(* CODESYS project BallSorting_student1.project

Project tree, tasks and I/O mapping:
  Device : CODESYS Control Win V3, 3S - Smart Software Solutions GmbH, version 3.5.17.10
    application Application
      libraries: Standard, * (System); Util, * (System); VisuDialogs, * (System)
      task MainTask (cyclic, interval t#20ms, priority 1) calls Model, PLC_PRG
      program Model [ST]: Initialization, Piston_Act, Interactions, Ball_Act, Output_Sensors
      data type PISTON
      visualisation Visualization
      data type BALL
      program PLC_PRG [SFC]: Alustus_active, Tunnistus_active, Lajittelu_active
  text list GlobalTextList
*)

// Device/Application/PISTON
TYPE PISTON :
STRUCT
	x	:REAL;	//Current x position of the piston's top-left corner with respect to 0,0 coordinates.
	xe	:REAL;	//Current x-axis elongation of the piston.
	y	:REAL;	//Current y position of the piston's top-left corner with respect to 0,0 coordinates.
	ye	:REAL;	//Current y-axis elongation of the piston.
	xf	:REAL;	//Maximum stroke of the piston in x-axis(mind the sign, a positive value indicates a stroke to the right).
	yf	:REAL;	//Maximum stroke of the piston in y-axis (mind the sign, a positive value indicates a stroke towards the bottom).
	xd	:BOOL;	//Indicates direction of stroke: TRUE = positive x; FALSE = negative x.
	se	:REAL;	//Eject speed of piston.
	sr	:REAL;	//Retract speed of piston.
END_STRUCT
END_TYPE

// Device/Application/BALL
TYPE BALL :
STRUCT
	x :REAL;		//Current x position of the ball assuming initial x position to be 0.
	xe :REAL;		//Velocity of the axis on the x-axis.
	y :REAL;		//Current y position of the ball assuming initial y position to be 0.
	ye :REAL;		//Velocity of the ball on the y-axis.
	rst :BOOL;		//Reset variable for the ball's y-axis velocity integrator.
	colour :DWORD;	//Colour of the ball. Should be written as: ball[x].colour := 16#00RRBBGG;
	m :INT;			//Material of the ball. A "1" represents a black ball, "2" corresponds to orange ball and "3" to grey ball.
END_STRUCT
END_TYPE

// Device/Application/Model
PROGRAM Model
VAR CONSTANT
	// Constant variables to be defined
	cycleTime :DWORD :=20;		//Base cycle time used in the PLC task (in ms).
	nBalls :INT := 9;			//Define number of balls.
	ballDiam :INT := 30;		//Define diameter of balls.
	ballXo :REAL :=320.0;		//Entrance x position of balls to visualization.
	ballYo :REAL :=0.0;			//Entrance y position of balls to visualization.
	nPistons :INT :=3;			//Number of pistons in the model.		
	speedBall :REAL :=5;		//Falling speed of balls.
END_VAR
VAR
	// Inputs array
	in :ARRAY[0..2] OF BOOL;
	// Outputs array
	out :ARRAY[0..5] OF BOOL;
	// Declare pistons array
	piston :ARRAY[0..nPistons-1] OF PISTON;
	// Declare balls array and their corresponding integrals
	ball :ARRAY[0..nBalls-1] OF BALL;
	doIntegral :ARRAY[0..nBalls-1] OF INTEGRAL;
	initialized :BOOL := FALSE;		//Value for setting the model with the initial conditions.
	b :INT;							//Used to store loop iterations during the program.
	bc :INT;						//Used to store loop iterations during the program.
	p :INT;							//Used to store loop iterations during the program.
	cycle :REAL;					//Stores the converted value to REAL of the cycle DWORD variable.
	ballInCanal :BOOL :=FALSE;		//Used for detecting whether a ball is present in the canal.
	ballOnSensor :BOOL :=FALSE;		//Used for detecting whether a ball is present in front of the material sensor.
	matBallOnSensor :INT :=0;		//Material of the ball present on the material sensor.
	laserPointer :REAL := - 400;	//Length of the laser line (maximum negative value represents maximum length of laser beam).
	autoMode :BOOL :=FALSE;			//Used to select between manual and automatic control.
	seed_1 :ULINT :=123;			//Used for the random number generator.
	seed_2 :ULINT :=456;
	tempInt :ULINT;
	random :REAL;
END_VAR

// Initialization, run once at the start of the PLC or when the "reset button" inside the visualization is pressed.
IF NOT initialized THEN
	Model.Initialization();
	initialized := TRUE;
END_IF

// Uncomment the following section once the variables "eject", "gate1" and "gate2" have been properly defined
// in your control program.

IF autoMode THEN
	in[0] := PLC_PRG.eject;
	in[1] := PLC_PRG.gate1;
	in[2] := PLC_PRG.gate2;
END_IF

// Four states of the system:
// State 1: update elongation of each piston.
Piston_Act();
// State 2: Update position of each ball.
Ball_Act();
// State 3: Determine interactions between pistons, balls and "solid bodies".
Interactions();
// State 4: Read information from model and update sensors' information.
Output_Sensors();

// Uncomment the following section once the variables "piston_in", "piston_out", "capacitive",
// "optical", "inductive" and "chute" have been properly defined in your control program.

PLC_PRG.piston_in := out[0];
PLC_PRG.piston_out := out[1];
PLC_PRG.capacitive := out[2];
PLC_PRG.optical := out[3];
PLC_PRG.inductive := out[4];
PLC_PRG.chute := out[5];

ACTION Initialization:
// Initialize pistons with correct values. Description of values can be found in "PISTON (STRUCT)".
// "piston[0]" corresponds to "Eject piston valve"
piston[0].xf := -60.0;
piston[0].xd := FALSE;
piston[0].y  := 177.0;
piston[0].se := 40;
piston[0].sr := 25;
piston[0].xe := 0;
// "piston[1]" corresponds to "Gate for 1. storage"
piston[1].xf := 30.0;
piston[1].xd := TRUE;
piston[1].se := 50;
piston[1].sr := 35;
piston[1].xe := 0;
// "piston[2]" corresponds to "Gate for 2. storage"
piston[2].xf := 30.0;
piston[2].xd := TRUE;
piston[2].se := 50;
piston[2].sr := 35;
piston[2].xe := 0;

// Reset inputs.
in[0] := FALSE;
in[1] := FALSE;
in[2] := FALSE;

// Initialize balls with correct initial position values and also reset any movement they might have.
FOR b:=0 TO nBalls - 1 DO
	ball[b].x := ballXo;	//"Entry point" of the balls to the system.
	ball[b].y := ballYo;
	ball[b].ye := 0.0;		//Reset speed in y axis.
	ball[b].xe := 0.0;		//Reset speed in x axis.
	ball[b].rst := TRUE;	//Reset the integral.
END_FOR

// Reset the material sensor.
out[2] :=FALSE;
out[3] :=FALSE;
out[4] :=FALSE;

// Define material of the balls.
// For this task, a random number generator is used which outputs a number between 0 and 1.
// Said number generator is based on the example of John D. Cook which can be found at:
// http://www.codeproject.com/Articles/25172/Simple-Random-Number-Generation
// Copyright (c) 2014, John D. Cook
// All rights reserved.
FOR b:=0 TO nBalls - 1 DO
	seed_1 := 36969* DWORD_TO_ULINT(( ULINT_TO_DWORD(seed_1) AND ULINT_TO_DWORD(65535)))+DWORD_TO_ULINT(SHR(ULINT_TO_DWORD(seed_1),16));
	seed_2 := 18000*DWORD_TO_ULINT(( ULINT_TO_DWORD(seed_2) AND ULINT_TO_DWORD(65535)))+ DWORD_TO_ULINT(SHR(ULINT_TO_DWORD(seed_2),16));
	tempInt := DWORD_TO_ULINT( SHL(ULINT_TO_DWORD(seed_2),16)) + seed_2;
	random := ULINT_TO_REAL(tempInt+1)*(2.328306435454494E-10);
	IF (random < 0.33) THEN
		ball[b].m := 1;
	END_IF
	IF (random >= 0.33) AND (random < 0.66) THEN
		ball[b].m := 2;
	END_IF
	IF (random >= 0.66) THEN
		ball[b].m := 3;
	END_IF
END_FOR

// Load each ball with the correct color value according to its material.
FOR b:=0 TO nBalls - 1 DO
	CASE ball[b].m OF
		1: ball[b].colour := 16#FF010101;	//Black ball.
		2: ball[b].colour := 16#FFFE9623;	//Orange ball.
		3: ball[b].colour := 16#FF666666;	//Grey ball.
	END_CASE
END_FOR
END_ACTION

ACTION Piston_Act:
// "cycleTime" is used as a scaling factor to determine the correct speed of the piston.
cycle :=DWORD_TO_REAL(cycleTime);

// Check each input and move pistons accordingly.
FOR p:=0 TO nPistons-1 DO
	IF in[p] AND NOT piston[p].xd AND (piston[p].xe > piston[p].xf) THEN
		piston[p].xe := piston[p].xe - (piston[p].se*cycle/1000.0);
		IF (piston[p].xe < piston[p].xf) THEN
			piston[p].xe := piston[p].xf;
		END_IF
	END_IF
	IF NOT in[p] AND NOT piston[p].xd AND (piston[p].xe < 0.0) THEN
		piston[p].xe := piston[p].xe + (piston[p].sr*cycle/1000.0);
		IF (piston[p].xe > 0.0) THEN
			piston[p].xe := 0.0;
		END_IF
	END_IF
	
	IF in[p] AND piston[p].xd AND (piston[p].xe < piston[p].xf) THEN
		piston[p].xe := piston[p].xe + (piston[p].se*cycle/1000.0);
		IF (piston[p].xe > piston[p].xf) THEN
			piston[p].xe := piston[p].xf;
		END_IF
	END_IF
	IF NOT in[p] AND piston[p].xd AND (piston[p].xe > 0.0) THEN
		piston[p].xe := piston[p].xe - (piston[p].sr*cycle/1000.0);
		IF (piston[p].xe < 0.0) THEN
			piston[p].xe := 0.0;
		END_IF
	END_IF
END_FOR
END_ACTION

ACTION Interactions:
piston[0].x := 350.0 + piston[0].xe;
piston[1].x := 260.0 + piston[1].xe;
piston[2].x := 260.0 + piston[2].xe;

FOR b:=0 TO (nBalls-1) DO
	//If any of the following conditions are true, the ball enters "falling" state (i.e. allow the integral to run). Conditions are position based
	//(i.e. check own position with respect to the position of the rest of elements in order to determine what the ball should do next).
	IF (ball[b].x > 319.9) AND (ball[b].y+ball[b].ye<(200.0-ballDiam)) AND (piston[0].x>342.0) THEN
		ball[b].rst :=FALSE;
	END_IF
	IF (ball[b].x > 319.9) AND (ball[b].y+ball[b].ye<(piston[0].y-ballDiam)) AND (piston[0].x<342.0) THEN
		ball[b].rst :=FALSE;
	END_IF
	IF (ball[b].x + ballDiam/2 < 285.1) AND (ball[b].y < 200.0) THEN
		ball[b].rst := FALSE;
	END_IF
	IF (ball[b].x + ballDiam < 290.1) AND (ball[b].y+ball[b].ye<570.0-ballDiam) THEN
		ball[b].x := 290.0 - ballDiam;
		ball[b].xe := 0.0;
		ball[b].rst := FALSE;
	END_IF
	
	//If any of the following conditions are true, the ball enters "waiting" state (i.e. reset integral).
	FOR bc:=0 TO (nBalls-1) DO
		IF (bc <> b) AND (ball[b].y < ball[bc].y) AND (ballDiam > SQRT(EXPT((ball[bc].y-(ball[b].y+ball[b].ye)),2)+EXPT((ball[bc].x-ball[b].x),2))) THEN
			ball[b].rst := TRUE;
			ball[b].ye := 0.0;
			ball[b].xe := 0.0;
		END_IF
	END_FOR
	IF (ball[b].x > 319.9) AND (ball[b].y + ball[b].ye > 200.0 - ballDiam) AND (ball[b].y < 200.0 - ballDiam) THEN
		ball[b].y := 200.0 - ballDiam;
		ball[b].rst := TRUE;
	END_IF
	IF (ball[b].x > 319.9) AND (ball[b].y + ball[b].ye > piston[0].y - ballDiam) AND (piston[0].x <= 342.0) AND (ball[b].y < piston[0].y-ballDiam) THEN
		ball[b].y := piston[0].y-ballDiam;
		ball[b].rst :=TRUE;
	END_IF
	IF (ball[b].y + ball[b].ye > 570.0 - ballDiam) THEN
		ball[b].xe := -(ball[b].ye);
		ball[b].rst := TRUE;
		ball[b].y := 570.0 - ballDiam;
	END_IF
	IF (ball[b].y + ball[b].ye > 310.0 - ballDiam) AND (ball[b].y < 310.0 - ballDiam) AND (piston[1].x > 260.0) THEN
		ball[b].y := 310.0 - ballDiam;
		ball[b].xe :=ball[b].ye*0.5;
		ball[b].rst :=TRUE;
		ball[b].ye :=0;
	END_IF
	IF (ball[b].y + ball[b].ye > 430.0-ballDiam) AND (ball[b].y < 430.0 - ballDiam) AND (piston[2].x > 260.0) THEN
		ball[b].y := 430.0 - ballDiam;
		ball[b].xe :=ball[b].ye*0.5;
		ball[b].rst :=TRUE;
		ball[b].ye :=0;
	END_IF
	
	// Always falling as long as reset input of the integral is false:
	IF NOT(ball[b].rst) THEN
		ball[b].y := ball[b].y+ball[b].ye;
	END_IF
	
	// Interactions for x axis of balls:
	IF (ball[b].y > 199.9 - ballDiam) AND (ball[b].y < 200.1-ballDiam) AND (piston[0].x < ball[b].x + ballDiam) THEN
		ball[b].x :=piston[0].x-ballDiam;
	END_IF
	IF (ball[b].y > 195.0 - ballDiam) AND (ball[b].y < 200.1-ballDiam) AND (ball[b].x + ballDiam/2 < 290.0) THEN
		ball[b].xe := ball[b].xe - speedBall*cycle/1000.0;
	END_IF
	IF (ball[b].y < 310.1 - ballDiam) AND (ball[b].y > 309.9 - ballDiam) AND (ball[b].x + ball[b].xe > 540.0 - ballDiam) THEN
		ball[b].x := 540 - ballDiam;
		ball[b].xe := 0.0;
	END_IF
	IF (ball[b].y < 430.1 - ballDiam) AND (ball[b].y > 429.9 - ballDiam) AND (ball[b].x + ball[b].xe > 540.0 - ballDiam) THEN
		ball[b].x := 540 - ballDiam;
		ball[b].xe := 0.0;
	END_IF
	IF (ball[b].y < 570.1 - ballDiam) AND (ball[b].y > 569.9 - ballDiam) AND (ball[b].x + ball[b].xe < 10.0) THEN
		ball[b].x := 10.0;
		ball[b].xe := 0.0;
	END_IF
	FOR bc:=0 TO (nBalls-1) DO
		IF (bc <> b) AND (ball[b].y + ballDiam >= ball[bc].y) AND (ball[b].y <= ball[bc].y) AND (ball[b].x+ball[b].xe+ballDiam > ball[bc].x)
		AND (ball[b].x < ball[bc].x) AND NOT(ball[bc].xe > 0.0) AND (ball[b].y > 200.0) THEN
			ball[b].xe := 0.0;
			ball[b].x := ball[bc].x - ballDiam;
		END_IF
		IF (bc <> b) AND (ball[b].y + ballDiam >= ball[bc].y) AND (ball[b].y <= ball[bc].y) AND (ball[b].x+ball[b].xe-ballDiam < ball[bc].x)
		AND (ball[b].x > ball[bc].x) AND NOT (ball[bc].xe > 0.0) AND (ball[b].y > 200.0)THEN
			ball[b].xe := 0.0;
			ball[b].x := ball[bc].x + ballDiam;
		END_IF
		IF (bc <> b) AND (ball[b].y >= ball[bc].y - 0.1) AND (ball[b].y <= ball[bc].y + 0.1) AND (ball[b].x < ball[bc].x + ballDiam)
		AND (ball[b].x > ball[bc].x) AND (ball[b].y < 200.0) AND (ball[bc].x>260.0) THEN
			ball[bc].x := ball[b].x-ballDiam;
		END_IF
		IF (bc <> b) AND (ball[b].y + ballDiam >= ball[bc].y) AND (ball[b].y <= ball[bc].y) AND (ball[b].x < ball[bc].x + ballDiam)
		AND (ball[b].x > ball[bc].x) AND (ball[b].y < 200.0) AND (ball[bc].x>260.0) THEN
			ball[bc].x := ball[bc].x-ball[b].ye;
		END_IF
	END_FOR
	//x position of a ball depends on its xe, except when this comes in conflict with solid bodies
	ball[b].x :=ball[b].x+ball[b].xe;
END_FOR
END_ACTION

ACTION Ball_Act:
FOR b:=0 TO (nBalls-1) DO
	doIntegral[b](IN:=speedBall,TM:=cycleTime,RESET:=ball[b].rst,OUT=>ball[b].ye);
END_FOR
END_ACTION

ACTION Output_Sensors:
FOR b:=0 TO nBalls - 1 DO
	// Check whether there is a ball over the sensor. In case there is, output its material.
	IF (ball[b].x > 315.0) AND (ball[b].y > (198.0-ballDiam)) AND (ball[b].y<(201.0-ballDiam)) THEN
		ballOnSensor := TRUE;
		matBallOnSensor := ball[b].m;
	END_IF
	// Check whether there is a ball in chute. If there is, the ball's position will determine the laser extension.
	IF ((ball[nBalls-1-b].x + ballDiam > 274.0) AND (ball[nBalls-1-b].x < 276.0)) AND (ball[nBalls-1-b].y > 199.9 - ballDiam) AND (ball[nBalls-1-b].y < 570.1 - ballDiam) THEN
		ballInCanal := TRUE;
		laserPointer := - 400 + (ball[nBalls-1-b].y - 185.0 + ballDiam);
	END_IF
END_FOR
// If any ball activated the sensor (i.e. it is present on the sensor), activate the correct sensors according to its material.
IF (ballOnSensor) THEN
	CASE matBallOnSensor OF
	1:  out[2] := TRUE;		//Black ball was detected.
		out[3] := FALSE;
		out[4] := FALSE;
		ballOnSensor := FALSE;
	2:  out[2] := TRUE;		//Orange ball was detected.
		out[3] := TRUE;
		out[4] := FALSE;
		ballOnSensor := FALSE;
	3:  out[2] := TRUE;		//Grey ball was detected.
		out[3] := TRUE;
		out[4] := TRUE;
		ballOnSensor := FALSE;
	END_CASE
ELSE						//If no ball is present on the sensors, reset them.
	out[2] := FALSE;
	out[3] := FALSE;
	out[4] := FALSE;
END_IF

// Output the information whether there is a ball in chute.
IF (ballInCanal) THEN
	out[5] := TRUE;
	ballInCanal := FALSE;
ELSE
	out[5] := FALSE;
	laserPointer := - 400.0;	
END_IF

// Check the "eject" piston position and activate corresponding sensor outputs if necessary.
IF (Model.piston[0].x > 349.0) THEN
	out[0] := TRUE;
ELSE		
	out[0] := FALSE;
END_IF
IF (Model.piston[0].x < 291.0) THEN
	out[1] := TRUE;
ELSE		
	out[1] := FALSE;
END_IF
END_ACTION

END_PROGRAM

// Device/Application/PLC_PRG
PROGRAM PLC_PRG
VAR_INPUT
	piston_in:BOOL;
	piston_out:BOOL;
	capacitive:BOOL;
	optical:BOOL;
	inductive:BOOL;
	chute:BOOL;
END_VAR
VAR_OUTPUT
	eject:BOOL;
	gate1:BOOL;
	gate2:BOOL;
END_VAR

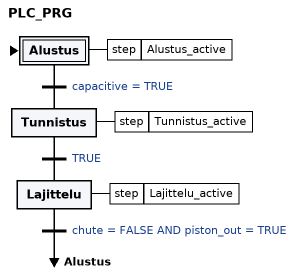
INITIAL_STEP Alustus:
    Alustus_active(N);  // step action
END_STEP
TRANSITION FROM Alustus TO Tunnistus
    := capacitive = TRUE;
END_TRANSITION
STEP Tunnistus:
    Tunnistus_active(N);  // step action
END_STEP
TRANSITION FROM Tunnistus TO Lajittelu
    := TRUE;
END_TRANSITION
STEP Lajittelu:
    Lajittelu_active(N);  // step action
END_STEP
TRANSITION FROM Lajittelu TO Alustus
    := chute = FALSE AND piston_out = TRUE;
END_TRANSITION

ACTION Alustus_active:
gate1 := FALSE;
gate2 := FALSE;
eject := FALSE;
END_ACTION

ACTION Tunnistus_active:
IF inductive = TRUE THEN;
	gate1 := TRUE;
ELSIF optical = TRUE AND inductive = FALSE THEN;
	gate2 := TRUE;	
END_IF
END_ACTION

ACTION Lajittelu_active:
eject := TRUE;
END_ACTION

END_PROGRAM

// Device/Application/Visualization
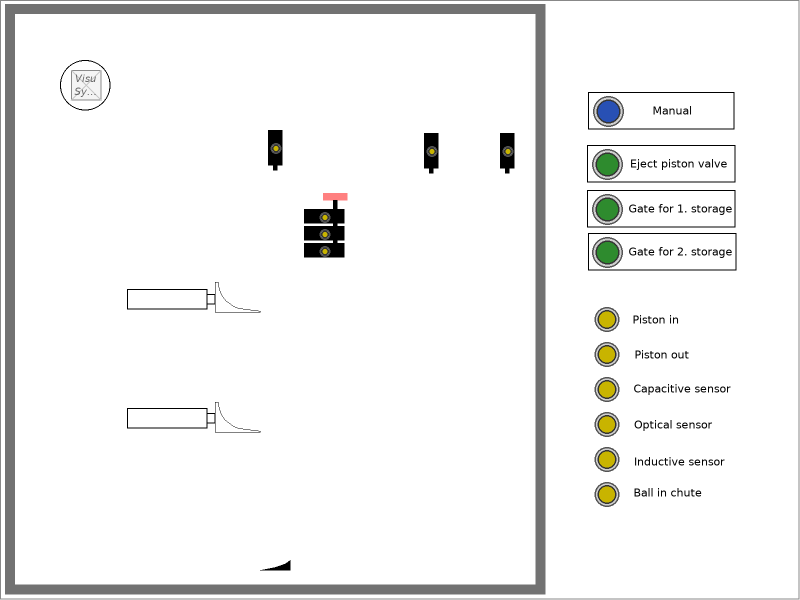
VISUALIZATION Visualization  // 800x600
    Rectangle (260,170 30x400)
    Line (275,570) (275,570)
        p2773130477: Model.laserPointer
    Rectangle (290,170 60x30)
    Rectangle (323,193 24x7)
    Rectangle (10,540 250x30)
    Rectangle (290,400 250x30)
    Rectangle (290,280 250x30)
    Rectangle (320,0 30x170)
    Ellipse (0,0 30x30), colour variable: Model.ball[0].colour
        p2738717112: Model.ball[0].y
        p3560616238: Model.ball[0].x
        p3450524324: Model.ball[0].colour
    Ellipse (0,0 30x30), colour variable: Model.ball[1].colour
        p2738717112: Model.ball[1].y
        p3560616238: Model.ball[1].x
        p3450524324: Model.ball[1].colour
    Ellipse (0,0 30x30), colour variable: Model.ball[2].colour
        p2738717112: Model.ball[2].y
        p3560616238: Model.ball[2].x
        p3450524324: Model.ball[2].colour
    Ellipse (0,0 30x30), colour variable: Model.ball[3].colour
        p2738717112: Model.ball[3].y
        p3560616238: Model.ball[3].x
        p3450524324: Model.ball[3].colour
    Ellipse (0,0 30x30), colour variable: Model.ball[4].colour
        p2738717112: Model.ball[4].y
        p3560616238: Model.ball[4].x
        p3450524324: Model.ball[4].colour
    Rectangle (268,130 14x35), tooltip "chute"
    Rectangle (273,165 4x5)
    Lamp1 (270,142 12x13), tooltip "chute", variable: Model.out[5], style: Lamp-Lamp1-Yellow
    Rectangle (304,209 40x14), tooltip "capacitive"
    Polygon (215,282) (215,312) (260,312) (260,311) (244,309) (238,308) (233,306) (229,303) (226,301) (222,296) (219,289) (218,282)
        p3560616238: Model.piston[1].xe
    Rectangle (179,294 36x10)
        p874137650: Model.piston[1].xe
    Rectangle (127,289 80x20), tooltip "gate1"
    Rectangle (410,180 70x10)
        p3528305787: Model.piston[0].xe
    Rectangle (350,177 60x16)
        p3560616238: Model.piston[0].xe
    Rectangle (418,173 100x24), tooltip "eject"
    Rectangle (424,133 14x35), tooltip "piston_out"
    Rectangle (500,133 14x35), tooltip "piston_in"
    Rectangle (429,168 4x5)
    Rectangle (505,168 4x5)
    Lamp1 (502,145 12x13), tooltip "piston_in", variable: Model.out[0], style: Lamp-Lamp1-Yellow
    Lamp1 (426,145 12x13), tooltip "piston_out", variable: Model.out[1], style: Lamp-Lamp1-Yellow
    Polygon (215,402) (215,432) (260,432) (260,431) (244,429) (238,428) (233,426) (229,423) (225,420) (221,414) (219,408) (218,402)
        p3560616238: Model.piston[2].xe
    Rectangle (179,413 36x10)
        p874137650: Model.piston[2].xe
    Rectangle (127,408 80x20), tooltip "gate2"
    Rectangle (333,200 4x9)
    Lamp1 (319,211 12x13), tooltip "capacitive", variable: Model.out[2], style: Lamp-Lamp1-Yellow
    Rectangle (304,226 40x14), tooltip "optical"
    Rectangle (333,220 4x9)
    Lamp1 (319,228 12x13), tooltip "optical", variable: Model.out[3], style: Lamp-Lamp1-Yellow
    Ellipse (0,0 30x30), colour variable: Model.ball[6].colour
        p2738717112: Model.ball[6].y
        p3560616238: Model.ball[6].x
        p3450524324: Model.ball[6].colour
    Ellipse (0,0 30x30), colour variable: Model.ball[7].colour
        p2738717112: Model.ball[7].y
        p3560616238: Model.ball[7].x
        p3450524324: Model.ball[7].colour
    Ellipse (0,0 30x30), colour variable: Model.ball[8].colour
        p2738717112: Model.ball[8].y
        p3560616238: Model.ball[8].x
        p3450524324: Model.ball[8].colour
    Ellipse (0,0 30x30), colour variable: Model.ball[5].colour
        p2738717112: Model.ball[5].y
        p3560616238: Model.ball[5].x
        p3450524324: Model.ball[5].colour
    Rectangle (304,243 40x14), tooltip "inductive"
    Rectangle (333,237 4x9)
    Lamp1 (319,245 12x13), tooltip "inductive", variable: Model.out[4], style: Lamp-Lamp1-Yellow
    Rectangle (320,0 30x45)
    Rectangle (0,0 60x60)
    Polygon (260,570) (290,570) (290,560) (286,563) (281,565) (275,567) (270,568) (265,569)
    Ellipse (60,60 50x50), tooltip "Reset"
    Image (71,70 30x30), tooltip "Reset", image: VisuSymbols.Symbols.ArrowHalfLeftLeft
        OnMouseDown: execute { Model.initialized := FALSE; }
    Lamp1 (591,94 35x35), variable: NOT(Model.autoMode), style: Lamp-Lamp1-Blue
    Label (628,96 89x30), "Manual"
    RoundedRectangle (588,92 146x37)
        OnMouseDown:  ToggleVariable=Model.autoMode
    Lamp1 (590,147 35x35), variable: Model.in[0], style: Lamp-Lamp1-Green
    Lamp1 (590,192 35x35), variable: Model.in[1], style: Lamp-Lamp1-Green
    Lamp1 (590,235 35x35), variable: Model.in[2], style: Lamp-Lamp1-Green
    Label (622,194 117x30), "Gate for 1. storage"
    Label (623,149 112x30), "Eject piston valve"
    Label (622,237 117x30), "Gate for 2. storage"
    RoundedRectangle (587,145 148x37)
        OnMouseDown:  ToggleVariable=Model.in[0]
    RoundedRectangle (587,190 148x37)
        OnMouseDown:  ToggleVariable=Model.in[1]
    RoundedRectangle (588,233 148x37)
        OnMouseDown:  ToggleVariable=Model.in[2]
    Lamp1 (593,305 28x29), variable: Model.out[0], style: Lamp-Lamp1-Yellow
    Lamp1 (593,340 28x29), variable: Model.out[1], style: Lamp-Lamp1-Yellow
    Lamp1 (593,480 28x29), variable: Model.out[5], style: Lamp-Lamp1-Yellow
    Lamp1 (593,410 28x29), variable: Model.out[3], style: Lamp-Lamp1-Yellow
    Lamp1 (593,375 28x29), variable: Model.out[2], style: Lamp-Lamp1-Yellow
    Lamp1 (593,445 28x29), variable: Model.out[4], style: Lamp-Lamp1-Yellow
    Label (611,307 90x26), "Piston in"
    Label (617,342 90x26), "Piston out"
    Label (626,376 112x26), "Capacitive sensor"
    Label (628,412 90x26), "Optical sensor"
    Label (627,449 105x26), "Inductive sensor"
    Label (623,480 90x26), "Ball in chute"
    Rectangle (5,4 540x590)
END_VISUALIZATION
